(* PLC project Device (Gm2xx), 未知 HydTechnology 0.1.0.0 *)
(* stored: creationDateTime 2026-08-13T17:06:11, modificationDateTime 2026-08-15T17:48:11 *)

(* __LUBAN_DATATYPE_TEXT_META__:{"comment":"","enum_value_comments":{"FTNone":"不滤波","FTLowPass":"低通滤波","FTMedian":"中值滤波","FTLimit":"限幅滤波","FTMovingAverage":"滑动窗口均值滤波"}} *)
TYPE E_FilterType : (FTNone, FTLowPass, FTMedian, FTLimit, FTMovingAverage, FTLowPassAndMovingAverage);
END_TYPE

TYPE ST_FilterConfig : STRUCT
  eType : E_FilterType;
  rParam1 : REAL := 0.1;  (* 通用参数1: *)
  uiParam2 : UINT := 3;  (* 通用参数2: - MovingAverage: 窗口大小(采样个数) *)
END_STRUCT;
END_TYPE

TYPE ST_SensorConfig : STRUCT
  rZeroVoltage : REAL;  (* 零点电压 *)
  rMaxVoltage : REAL;  (* 最大电压 *)
  rRange : REAL;  (* 量程 (例如: 10.0 MPa 或 500.0 mm) *)
END_STRUCT;
END_TYPE

TYPE E_AxisState : (eInit, eReady, eIdle, eBusy, eDone, eStopping, eStopped, eEmergencyStop, eError);
END_TYPE

TYPE E_AxisMode : (eNone, ePosition, eVelocity, ePressure);
END_TYPE

TYPE E_PumpPolicy : (eMotionDefault, eProcessPriority);
END_TYPE

TYPE E_ProcessStep : (eStepIdle, eStepSegment1, eStepSegment2, eStepPressure, eStepDwell, eStepDone, eStepError);
END_TYPE

TYPE ST_AxisStatus : STRUCT
  eState : E_AxisState;
  bEnabled : BOOL;
  bBusy : BOOL;
  bDone : BOOL;
  bError : BOOL;
  udiErrorID : UDINT;
  rActualPosition : LREAL;
  rActualVelocity : LREAL;
  rActualPressure : REAL;
END_STRUCT;
END_TYPE

TYPE ST_HydPumpStatus : STRUCT
  rPumpSpeed : REAL;
  bConflict : BOOL;
  bBusy : BOOL;
  bDone : BOOL;
  bError : BOOL;
  wErrorID : WORD;
  bCycleReentry : BOOL;
END_STRUCT;
END_TYPE

TYPE ST_HydAxisRef : STRUCT
  bFunBlockStart : BOOL;  (* FB：启动信号 *)
  bStart : BOOL;  (* 轴：启动信号 *)
  bStop : BOOL;  (* 轴：停止信号 *)
  uiDir : UINT;  (* 轴：设定方向 *)
  udiPos : UDINT;  (* 轴：设定位置 *)
  uiSpd : UINT;  (* 轴：设定速度 *)
  uiEndSpd : UINT;  (* 轴：设定结束速度 *)
  uiPres : UINT;  (* 轴：设定压力 *)
  rPosition : REAL;  (* 轴：反馈位置 *)
  rVeloctity : REAL;  (* 轴：反馈速度 *)
  rPerssure : REAL;  (* 轴：反馈压力 *)
  rFlow : REAL;  (* 轴：反馈流量 *)
  iStep : INT;  (* 轴：反馈当前步号 *)
  rActPressure : REAL;
  rActPosition : REAL;
  rActVelocity : REAL;
  rMaxSpeed : REAL;  (* 当前轴的最大速度设定 *)
  rMaxSpeedExtend : REAL;  (* 液压轴伸出侧最大速度 *)
  rMaxSpeedRetract : REAL;  (* 液压轴缩回侧最大速度 *)
  rVelToFlowGain : REAL := 0.2;  (* 速度流量增益 *)
  rCylinderExtendArea : REAL := 0;  (* 油缸伸出腔有效面积mm2 *)
  rCylinderRetractArea : REAL := 0;  (* 油缸缩回腔有效面积mm2 *)
  iTypePressurePID : SINT := 4;  (* 压力闭环类型 *)
  iAxisID : SINT := -1;  (* 轴索引 *)
  iMechanismType : SINT := 0;  (* 机械运动学类型 *)
END_STRUCT;
END_TYPE

INTERFACE ?
END_INTERFACE

INTERFACE ?
END_INTERFACE

FUNCTION_BLOCK FB_LimitFilter
  VAR_INPUT
    rInput : REAL;
    rMaxDiff : REAL;  (* RC:[最大允许变化幅值] *)
  END_VAR
  VAR_OUTPUT
    rOutput : REAL;
  END_VAR
  VAR
    bFirstRun : BOOL := TRUE;
  END_VAR

            IF bFirstRun THEN
    rOutput := rInput;
    bFirstRun := FALSE;
ELSE
    IF ABS(rInput - rOutput) > rMaxDiff THEN
        rOutput := rOutput; // 超出限幅，保持上次值不变
    ELSE
        rOutput := rInput;  // 正常范围内，更新
    END_IF;
END_IF;
          
END_FUNCTION_BLOCK

FUNCTION_BLOCK FB_LowPassFilter
  VAR_INPUT
    rInput : REAL;
    rAlpha : REAL;  (* RC:[滤波系数 (0.0~1.0)] *)
  END_VAR
  VAR_OUTPUT
    rOutput : REAL;
  END_VAR
  VAR
    bFirstRun : BOOL := TRUE;
  END_VAR

            IF bFirstRun THEN
    rOutput := rInput;
    bFirstRun := FALSE;
ELSE
    rOutput := rOutput + rAlpha * (rInput - rOutput);
END_IF;
          
END_FUNCTION_BLOCK

FUNCTION_BLOCK FB_MedianFilter
  VAR_INPUT
    rInput : REAL;
  END_VAR
  VAR_OUTPUT
    rOutput : REAL;
  END_VAR
  VAR
    aBuffer : ARRAY[1..3] OF REAL;
    iPtr : INT := 1;
    aSort : ARRAY[1..3] OF REAL;
    i : INT;
    j : INT;
    rTemp : REAL;
  END_VAR

            // 存入循环缓冲区
aBuffer[iPtr] := rInput;
iPtr := iPtr + 1;
IF iPtr > 3 THEN iPtr := 1; END_IF;

// 复制到排序数组
aSort := aBuffer;

// 冒泡排序 (3个元素，最多3次比较)
FOR i := 1 TO 2 DO
    FOR j := 1 TO (3 - i) DO
        IF aSort[j] > aSort[j+1] THEN
            rTemp := aSort[j];
            aSort[j] := aSort[j+1];
            aSort[j+1] := rTemp;
        END_IF;
    END_FOR;
END_FOR;

// 取中间值
rOutput := aSort[2];
          
END_FUNCTION_BLOCK

FUNCTION_BLOCK FB_MovingAverageFilter
  VAR_INPUT
    rInput : REAL;
    uiSize : UINT := 1;  (* RC:[窗口大小] *)
  END_VAR
  VAR_OUTPUT
    rOutput : REAL;
  END_VAR
  VAR
    aBuffer : ARRAY[1..100] OF REAL;  (* RC:[最大支持100个数据窗口] *)
    iPtr : UINT := 1;
    rSum : REAL;
    iCount : INT := 0;
    i : UINT;
  END_VAR

            IF uiSize > 100 THEN uiSize := 100; END_IF;
IF uiSize = 0 THEN uiSize := 1; END_IF;

// 更新缓冲区
aBuffer[iPtr] := rInput;
iPtr := iPtr + 1;
IF iPtr > uiSize THEN iPtr := 1; END_IF;

// 求和计算平均值
rSum := 0.0;
FOR i := 1 TO uiSize DO
    rSum := rSum + aBuffer[i];
END_FOR;

rOutput := rSum / UINT_TO_REAL(uiSize);
          
END_FUNCTION_BLOCK

FUNCTION_BLOCK FB_PositionSensor
  VAR_INPUT
    uiRawADC : UINT;
  END_VAR
  VAR_OUTPUT
    rActualValue : REAL;  (* RC:[滤波后的最终输出] *)
    rActualValueDeriv : REAL;
    rRawValue : REAL;  (* RC:[未滤波的原始转换值 (便于调试对比)] *)
    bAlarm : BOOL;
  END_VAR
  VAR
    stConfig : ST_SensorConfig;
    stFilterCfg : ST_FilterConfig;
    rVoltage : REAL;
    fbLowPass : FB_LowPassFilter;  (* UC:[实例化滤波器] *)
    fbLimit : FB_LimitFilter;
    fbMedian : FB_MedianFilter;
    fbMovingAvg : FB_MovingAverageFilter;
    bUpperLimit : BOOL;  (* UC:[可以在此扩展位置传感器特有的变量，例如：位置限位报警] *)
    bLowerLimit : BOOL;
    rLastActualValue : REAL;
  END_VAR
  VAR CONSTANT
    cADC_MAX : REAL := 65535.0;
    cVOLTAGE_MAX : REAL := 10.0;
    cTCycle : REAL := 0.001;
  END_VAR

            // --- 主逻辑 ---

// 1. 物理量转换
IF (stConfig.rMaxVoltage - stConfig.rZeroVoltage) <= 0.0 THEN
    bAlarm := TRUE;
    rRawValue := 0.0;
ELSE
    bAlarm := FALSE;
    rRawValue := (UINT_TO_REAL(uiRawADC) - stConfig.rZeroVoltage) / 
                 (stConfig.rMaxVoltage - stConfig.rZeroVoltage) * 
                 stConfig.rRange;
    rRawValue := LIMIT(0.0,rRawValue,stConfig.rRange);
END_IF;

// 2. 滤波处理链 (采用单一配置切换，若需组合可级联调用)
CASE stFilterCfg.eType OF
    FTLowPass:
        fbLowPass(rInput := rRawValue, rAlpha := stFilterCfg.rParam1);
        rActualValue := fbLowPass.rOutput;
        
    FTLimit:
        fbLimit(rInput := rRawValue, rMaxDiff := stFilterCfg.rParam1);
        rActualValue := fbLimit.rOutput;
        
    FTMedian:
        fbMedian(rInput := rRawValue);
        rActualValue := fbMedian.rOutput;
        
    FTMovingAverage:
        fbMovingAvg(rInput := rRawValue, uiSize := stFilterCfg.uiParam2);
        rActualValue := fbMovingAvg.rOutput;
    
    FTLowPassAndMovingAverage:
        fbLowPass(rInput := rRawValue, rAlpha := stFilterCfg.rParam1);
        fbMovingAvg(rInput :=  fbLowPass.rOutput, uiSize := stFilterCfg.uiParam2);
        rActualValue := fbMovingAvg.rOutput;     
      
ELSE
    // None: 不滤波
    rActualValue := rRawValue;
END_CASE;

rActualValueDeriv := ( rActualValue - rLastActualValue )/cTCycle;
rLastActualValue := rActualValue;
          

METHOD Init : BOOL
  VAR_INPUT
    rZero : REAL;
    rMax : REAL;
    rRng : REAL;
  END_VAR
                  stConfig.rZeroVoltage := rZero;
stConfig.rMaxVoltage  := rMax;
stConfig.rRange       := rRng;
Init := TRUE;
                
END_METHOD

METHOD SetFilter : BOOL
  VAR_INPUT
    eType : E_FilterType;
    rParam1 : REAL;
    uiParam2 : UINT;
  END_VAR
                  stFilterCfg.eType := eType;
stFilterCfg.rParam1 := rParam1;
stFilterCfg.uiParam2 := uiParam2;
SetFilter := TRUE;
                
END_METHOD
END_FUNCTION_BLOCK

FUNCTION_BLOCK FB_PressureSensor
  VAR_INPUT
    uiRawADC : UINT;
  END_VAR
  VAR_OUTPUT
    rActualValue : REAL;  (* RC:[滤波后的最终输出] *)
    rRawValue : REAL;  (* RC:[未滤波的原始转换值 (便于调试对比)] *)
    bAlarm : BOOL;
  END_VAR
  VAR
    stConfig : ST_SensorConfig;
    stFilterCfg : ST_FilterConfig;
    fbLowPass : FB_LowPassFilter;  (* UC:[实例化滤波器] *)
    fbLimit : FB_LimitFilter;
    fbMedian : FB_MedianFilter;
    fbMovingAvg : FB_MovingAverageFilter;
  END_VAR
  VAR CONSTANT
    cADC_MAX : REAL := 65535.0;
    cVOLTAGE_MAX : REAL := 10.0;
  END_VAR

            
// 1. 物理量转换
IF (stConfig.rMaxVoltage - stConfig.rZeroVoltage) <= 0.0 THEN
    bAlarm := TRUE;
    rRawValue := 0.0;
ELSE
    bAlarm := FALSE;
    rRawValue := (UINT_TO_REAL(uiRawADC) - stConfig.rZeroVoltage) / 
                 (stConfig.rMaxVoltage - stConfig.rZeroVoltage) * 
                 stConfig.rRange;
    rRawValue := LIMIT(0.0,rRawValue,stConfig.rRange);

END_IF;

// 2. 滤波处理链 (采用单一配置切换，若需组合可级联调用)
CASE stFilterCfg.eType OF
    FTLowPass:
        fbLowPass(rInput := rRawValue, rAlpha := stFilterCfg.rParam1);
        rActualValue := fbLowPass.rOutput;
        
    FTLimit:
        fbLimit(rInput := rRawValue, rMaxDiff := stFilterCfg.rParam1);
        rActualValue := fbLimit.rOutput;
        
    FTMedian:
        fbMedian(rInput := rRawValue);
        rActualValue := fbMedian.rOutput;
        
    FTMovingAverage:
        fbMovingAvg(rInput := rRawValue, uiSize := stFilterCfg.uiParam2);
        rActualValue := fbMovingAvg.rOutput;

    FTLowPassAndMovingAverage:
        fbLowPass(rInput := rRawValue, rAlpha := stFilterCfg.rParam1);
        fbMovingAvg(rInput :=  fbLowPass.rOutput, uiSize := stFilterCfg.uiParam2);
        rActualValue := fbMovingAvg.rOutput;  
        
ELSE
    // None: 不滤波
    rActualValue := rRawValue;
END_CASE;
          

METHOD Init : BOOL
  VAR_INPUT
    rZero : REAL;
    rMax : REAL;
    rRng : REAL;
  END_VAR
                  stConfig.rZeroVoltage := rZero;
stConfig.rMaxVoltage  := rMax;
stConfig.rRange       := rRng;
Init := TRUE;
                
END_METHOD

METHOD SetFilter : BOOL
  VAR_INPUT
    eType : E_FilterType;
    rParam1 : REAL;
    uiParam2 : UINT;
  END_VAR
                  stFilterCfg.eType := eType;
stFilterCfg.rParam1 := rParam1;
stFilterCfg.uiParam2 := uiParam2;
SetFilter := TRUE;
                
END_METHOD
END_FUNCTION_BLOCK

FUNCTION_BLOCK FB_ServoControl
  VAR_INPUT
    StartMotor : BOOL;  (* RC:[TRUE: 使能并启动电机, FALSE: 减速停止并断使能] *)
    SetVelCmd : REAL;
    FlowRateLimit : UINT;
    uiMaxMotorSpeed : UINT;
    EnSimulation : BOOL;
    SelfLearn : BOOL;
    UsePlanner : BOOL;
    tcycle : REAL := 0.001;
  END_VAR
  VAR_OUTPUT
    ActSpeedRPM : UINT;
    ActPressBAR : UINT;
    outErrorID : UINT;
    Status : UINT;
    ActMotorPos : UINT;  (* RC:[360deg] *)
    ActTorquePercent : UINT;  (* RC:[0.1%] *)
  END_VAR
  VAR
    STATE_INIT : DINT := 0;  (* UC:[--- 状态机常量 ---] *)
    STATE_READ_SDO1 : DINT := 1;
    STATE_READ_SDO2 : DINT := 2;
    STATE_WRITE_PARAM : DINT := 10;
    STATE_SELFLEARN : DINT := 20;
    STATE_SET_MODE : DINT := 30;
    STATE_IDLE : DINT := 40;  (* RC:[等待使能] *)
    STATE_RUNNING : DINT := 50;  (* RC:[速度运行中] *)
    STATE_STOPPING : DINT := 60;  (* RC:[减速停机中] *)
    STATE_ERROR : DINT := 99;
    iState : DINT := 0;  (* UC:[--- 内部变量 ---] *)
    fbDelay : TON;  (* UC:[--- 功能块实例 ---] *)
    fbPower : MC_Power;
    fbFollowVel : SMC_FollowVelocity;
    fbSetPar : MC_WriteParameter;
    fbSetBoolPar : MC_WriteBoolParameter;
    fbReset : MC_Reset;
    fbModeCtrl : MC_SetControllerMode;
    fbReadVel : MC_ReadActualVelocity;
    fbReadPos : MC_ReadActualPosition;
    fbReadTor : MC_ReadActualTorque;
    fbSDORead : PorgaSDOUpload;
    fbStartMotorSelfLearn : StartMotorSelfLearn;
    nAxisRef : AXIS_REF := 0;
    bPowerCmd : BOOL := FALSE;  (* RC:[映射到 MC_Power.Enable] UC:[--- 运动控制核心指令标志位 ---] *)
    bMoveCmd : BOOL := FALSE;  (* RC:[映射到 SMC_FollowVelocity.Execute] *)
    dfSetVel : LREAL := 0.0;  (* RC:[映射到 SMC_FollowVelocity.Velocity] *)
    Error : BOOL := 0;  (* UC:[--- 数据与参数 ---] *)
    ErrorID : WORD := 0;
    MaxVel : LREAL := 12000.0;
    MaxAcc : LREAL := 12000.0;
    MaxJerk : LREAL := 12000.0;
    dfActVel : LREAL := 0.01;
    dfActVelFb : LREAL := 0.01;
    dfActPosFb : LREAL := 0.01;
    dfActTor : LREAL := 0.01;
    dir : LREAL := -1.0;
    fMotorSpeedLimit : LREAL := 0.0;
    fSetVel : LREAL := 0.0;
    dfMinVel : LREAL := -100.0;
    wNumBitEnc : UDINT := 0;
    wTempVar : UDINT := 0;
    dfResolutionEnc : LREAL := 0.0;
    wDirRotate : WORD := 0;
    arMotorParam : PAR_WORD_ARRAY := [3333, 107, 380, 20, 200, 5000, 100, 0, 0, 0];
  END_VAR

            
(*=====================================================================*)
(*               1. 运算与条件准备 (每周期执行)                          *)
(*=====================================================================*)

// 速度与压力设定值计算 (仅在初始化完成后计算)
IF iState >= STATE_IDLE THEN

    MaxVel  := UINT_TO_LREAL(uiMaxMotorSpeed) * (360.0/60.0); 
    MaxAcc  := 2.0 * MaxVel;
    MaxJerk := 3.0 * MaxVel;
    fMotorSpeedLimit := UINT_TO_LREAL(uiMaxMotorSpeed) * LIMIT(0, FlowRateLimit, 1000) * 0.001;
    fSetVel := REAL_TO_LREAL(SetVelCmd);
    fSetVel := LIMIT( dfMinVel, fSetVel, fMotorSpeedLimit );     
    
    fSetVel := fSetVel * dir;
END_IF;

// 使能命令统一映射 (PowerEnable 掌控全局)
bPowerCmd := StartMotor AND (iState >= STATE_IDLE);

(*=====================================================================*)
(*               2. 状态机 (仅控制逻辑流转与指令赋值)                     *)
(*=====================================================================*)

CASE iState OF

    0: // 0: 初始化IP与SDO1
        
        fbSDORead( Axis := nAxisRef, Execute := TRUE, Index := 19, Size := 1 );
        iState := STATE_READ_SDO1;

    1: // 1: 等待SDO1读取完成 (异步处理)
        fbSDORead( Axis := nAxisRef, Execute := TRUE, Index := 19, Size := 1 );
        IF fbSDORead.Done THEN
            wNumBitEnc := WORD_TO_UDINT( fbSDORead.ValueArray[1] );
            IF wNumBitEnc > 1 AND wNumBitEnc < 60 THEN
                wTempVar := SHL(1, wNumBitEnc);
            ELSE
                wTempVar := SHL(1, 12);
            END_IF;
            dfResolutionEnc := UDINT_TO_LREAL(wTempVar);
            fbSDORead( Execute := FALSE );
            fbSDORead( Axis := nAxisRef, Execute := TRUE, Index := 106, Size := 1 );
            iState := STATE_READ_SDO2;
        END_IF;

    2: // 2: 等待SDO2读取完成
        fbSDORead( Axis := nAxisRef, Execute := TRUE, Index := 106, Size := 1 );
        IF fbSDORead.Done THEN
            wDirRotate := fbSDORead.ValueArray[1];
            fbSDORead( Execute := FALSE );
            iState := STATE_WRITE_PARAM;
        END_IF;

    10: // 10: 写入参数与仿真设置
        fbSetPar(Axis := nAxisRef, Execute := TRUE, ParameterNumber:= 1003, Value := dfResolutionEnc);  // 4096
        fbSetBoolPar(Axis := nAxisRef, Execute := TRUE, ParameterNumber:= 1000, Value := EnSimulation);
        IF fbSetPar.Done AND fbSetBoolPar.Done THEN
            fbSetPar(Execute := FALSE);
            fbSetBoolPar(Execute := FALSE);
            fbReset( Axis := nAxisRef, Execute := FALSE );
            fbStartMotorSelfLearn( Axis := nAxisRef, Execute := FALSE );
            iState := STATE_SELFLEARN;
        END_IF;

    20: // 20: 自学习
        IF SelfLearn THEN
            fbStartMotorSelfLearn( Axis := nAxisRef, Execute := TRUE,
                                   ResetServoParam := TRUE, WriteServoParam := TRUE,
                                   MotorLearn := TRUE, ParameterArray := arMotorParam );
            IF fbStartMotorSelfLearn.Done THEN
                fbStartMotorSelfLearn(Execute := FALSE);
                iState := STATE_SET_MODE;
            END_IF;
        ELSE
            iState := STATE_SET_MODE;
        END_IF;

    30: // 30: 设置控制模式
        fbModeCtrl(Axis := nAxisRef, Execute := TRUE, ControllerMode := mcFollowVelocity, ExecutionMode := mcImmediately);
        IF fbModeCtrl.Done THEN
            fbModeCtrl(Execute := FALSE);
            iState := STATE_IDLE;
        END_IF;

    40: // 40: 待机状态 (等待 PowerEnable)
        bMoveCmd := FALSE;
        dfSetVel := 0.0;
        // 核心逻辑：给使能 且 电机已成功使能，则立即启动速度控制
        IF StartMotor AND fbPower.Status THEN
            iState := STATE_RUNNING;
        END_IF;

    50: // 50: 速度运行中
        bMoveCmd := TRUE;
        dfSetVel := fSetVel * (360.0/60.0); // RPM 转换 UU/s

        // 核心逻辑：一旦失去使能信号，立即进入减速停机
        IF NOT StartMotor THEN
            iState := STATE_STOPPING;
        END_IF;

    60: // 60: 减速停机中
        bMoveCmd := TRUE;  // 保持速度块 Execute，以控制减速曲线
        dfSetVel := 0.0;   // 目标速度设为 0

        // 减速中途，如果使能信号恢复，立即恢复运行
        IF StartMotor THEN
            fbDelay(IN := FALSE); // 清除停机定时器
            iState := STATE_RUNNING;
        ELSE
            // 速度低于阈值开始计时，若速度反弹则自动复位定时器
            fbDelay(IN := ABS(dfActVel) < 5.0, PT := TIME#1S);
            IF fbDelay.Q THEN
                bMoveCmd := FALSE;    // 停机完成，撤销速度控制命令
                fbDelay(IN := FALSE); // 复位定时器
                iState := STATE_IDLE; // 回到待机 (bPowerCmd随之变FALSE，自动断使能)
            END_IF;
        END_IF;

    99: // 99: 错误状态
        Error := TRUE;
        bMoveCmd := FALSE;

END_CASE;

(*=====================================================================*)
(*          3. 统一调用 PLCopen 功能块 (严格遵循规范，每周期执行)         *)
(*=====================================================================*)
//(*  更新液压系统模型 *)
//hydraulic_sys.motorvelocity := SetVelCmd;
//hydraulic_sys.tcycle := tcycle;
//hydraulic_sys.knum := 5.4;   // 4.2, 1.162, 5.4
//hydraulic_sys.ttau := 1.0;   // 0.4, 0.171, 1.0 
//hydraulic_sys.delaytime := 0.0;  // 1.0 max , 0.438
//hydraulic_sys();

// 使能控制
fbPower( Axis := nAxisRef, Enable := bPowerCmd, EnablePositive := TRUE, EnableNegative := TRUE);

// 速度跟随控制
fbFollowVel( Axis := nAxisRef, Execute := bMoveCmd, Velocity := dfSetVel);

// 反馈读取 (进入Idle后即开始读取，保证状态监控连续性)
IF iState >= STATE_IDLE THEN
    fbReadVel( Axis := nAxisRef, Enable := TRUE, Velocity => dfActVel, VelocityFeedback => dfActVelFb);
    fbReadPos( Axis := nAxisRef, Enable := TRUE, Position => dfActPosFb );
    fbReadTor( Axis := nAxisRef, Enable := TRUE, Torque   => dfActTor);  
END_IF;

// 错误捕获 (从运动功能块中提取错误)
IF fbFollowVel.Error THEN
    ErrorID := fbFollowVel.ErrorID;
    iState := STATE_ERROR;
END_IF;

(*=====================================================================*)
(*                      4. 输出映射                                     *)
(*=====================================================================*)

Status          := DINT_TO_UINT(iState);
outErrorID      := ErrorID;
ActSpeedRPM := DINT_TO_UINT( LREAL_TO_DINT(dfActVel*60.0/360.0) );
ActTorquePercent := DINT_TO_UINT( LREAL_TO_DINT(dfActTor) );
          
END_FUNCTION_BLOCK

FUNCTION_BLOCK FB_HydAxis
  VAR_IN_OUT
    stHydAxisRef : ST_HydAxisRef;
  END_VAR
  VAR_INPUT
    bStart : BOOL;
    bStop : BOOL;
    bEStop : BOOL;
    bReset : BOOL;
    uiDir : UINT;  (* RC:[0:无效 1:正向 2:反向] *)
    uiMode : UINT;  (* RC:[0:无效 1:位置 2:速度 3:压力] *)
    uiPres : UINT;
    uiSpd : UINT;
    uiEndSpd : UINT;
    udiPos : UDINT;
    uiForce : UINT;
    uiAcc : UINT;
    uiDec : UINT;
    uiJerk : UINT;
    kkk : UINT;
  END_VAR
  VAR_OUTPUT
    bBusy : BOOL;  (* RC:[TRUE=轴层当前仍保持有效执行命令] *)
    bDone : BOOL; // TRUE=位置模式下到达InEndVelocity(段结束); TRUE=非位置模式下指令执行完成且空闲;
    bInVelocity : BOOL;
    bInPressure : BOOL;
    bAlarm : BOOL;
    dwAlarmID : DWORD;
  END_VAR
  VAR
    iStep : INT;  (* RC:[0初始化, 10空闲, 100运行, 105运行过渡(产生脉冲), 200停止, 300急停, 400复位, 900报警] *)
    fbCreate : HYD_CreateMotion;
    fbMoveContAbs : HYD_MoveContinuousAbsolute;
    fbMoveVel : HYD_MoveVelocity;
    fbPresHdl : HYD_PressureHandle;
    fbStop : HYD_Stop;
    fbEStop : HYD_Stop;
    fbReset : HYD_Reset;
    fbReadFB : HYD_ReadSimFeedback;
    fbHYD_WriteParameter : HYD_WriteParameter;
    fbHYD_SetAxisFeedback : HYD_SetAxisFeedback;
    fbCalcMaxSpeed : FB_CalcAxisMaxSpeed;
    siAxisId : SINT;
    rTrigStart : R_TRIG;
    rTrigStop : R_TRIG;
    rTrigEStop : R_TRIG;
    rTrigReset : R_TRIG;
    rTrigDone : R_TRIG;
    uiActiveMode : UINT;  (* RC:[当前执行模式 (1:Pos, 2:Vel, 3:Pres)] *)
    bCmdExecute : BOOL;  (* RC:[统一控制当前活跃模式的 Execute 引脚] *)
    iDir : SINT;
    rPos : REAL;
    rVel : REAL;
    rEndVel : REAL;  (* RC:[终点速度] *)
    rPres : REAL;
    rAcc : REAL;
    rDec : REAL;
    rJerk : REAL;
    bFBError : BOOL;
    wFBErrorID : WORD;
    iDoneCnt : INT := 0;
    rMaxSpeed : REAL;  (* RC:[单位mm/s] *)
    rPosition : REAL;
    rVeloctity : REAL;
    rFlow : REAL;
    rPerssure : REAL;
    rCycle : REAL;
  END_VAR

            // 仅作监视调试使用
// 轴：启动信号、停止信号、设定位置、设定速度、设定结束速度、设定压力
stHydAxisRef.bStart := bStart;
stHydAxisRef.bStop := bStop;
stHydAxisRef.uiDir := uiDir;
stHydAxisRef.udiPos := udiPos;
stHydAxisRef.uiSpd := uiSpd;
stHydAxisRef.uiEndSpd := uiEndSpd;
stHydAxisRef.uiPres := uiPres;

//--- 1. 边沿检测 & 参数映射 ---
rTrigStart(CLK := bStart);
rTrigStop(CLK := bStop);
rTrigEStop(CLK := bEStop);
rTrigReset(CLK := bReset);
// 将Done检测移出CASE，确保全周期扫描，不错过InEndVelocity的上升沿
rTrigDone(CLK := fbMoveContAbs.InEndVelocity); 

rMaxSpeed := stHydAxisRef.rMaxSpeed;

//IF stHydAxisRef.rCylinderExtendArea > 0.0 AND stHydAxisRef.rCylinderRetractArea > 0.0 THEN
//  IF uiDir = 1 THEN
//    rMaxSpeed := stHydAxisRef.rMaxSpeedExtend;
//  ELSE
//    rMaxSpeed := stHydAxisRef.rMaxSpeedRetract;
//  END_IF;
//END_IF;

rPres := MAX(UINT_TO_REAL(uiPres), 0.0)*0.1;   //压力设定
rVel  := UINT_TO_REAL(uiSpd)*0.1*0.01*rMaxSpeed;  //速度设定
rEndVel := UINT_TO_REAL(uiEndSpd)*0.1*0.01*rMaxSpeed;  //终点速度，连续轨迹关键：设定终点速度等于最大速度，实现"到位不停车"或平滑过渡
rPos  := UDINT_TO_REAL(udiPos)*0.01;  //位置设定


IF uiAcc = 0 THEN rAcc := 200; ELSE rAcc  := rMaxSpeed/UINT_TO_REAL(uiAcc)*1000; END_IF;  
IF uiDec = 0 THEN rDec := 200; ELSE rDec  := rMaxSpeed/UINT_TO_REAL(uiDec)*1000; END_IF;  
IF uiJerk = 0 THEN rJerk := 0; ELSE rJerk := rMaxSpeed/UINT_TO_REAL(uiJerk); END_IF;

iDir := uiDir;  
//--- 2. 状态机主逻辑 ---
CASE iStep OF

    0: // 初始化
        fbCreate(USE_SIMULATION := 0, MECHANISM_TYPE:= stHydAxisRef.iMechanismType);
        IF fbCreate.DONE THEN
            siAxisId := fbCreate.AXISID;
            stHydAxisRef.iAxisID := siAxisId;
            SetVelocityToFlowGain(stHydAxisRef.rVelToFlowGain);
            SetPidType( SINT_TO_REAL(stHydAxisRef.iTypePressurePID) );
            SetCylinderConfig(stHydAxisRef.rCylinderExtendArea, stHydAxisRef.rCylinderRetractArea );
            fbCalcMaxSpeed(stHydAxisRef.rCylinderExtendArea, stHydAxisRef.rCylinderRetractArea, 1800, 50, stHydAxisRef.iMechanismType );
            stHydAxisRef.rMaxSpeedExtend  := fbCalcMaxSpeed.rMaxSpeedExtend;
            stHydAxisRef.rMaxSpeedRetract := fbCalcMaxSpeed.rMaxSpeedRetract;
            iStep := 10;
        ELSIF fbCreate.ERROR THEN
            bAlarm := TRUE; dwAlarmID := 16#00000001; iStep := 900;
        END_IF;

    10: // 空闲
        bCmdExecute := FALSE; 
        bDone := FALSE; // 重置完成信号
        IF rTrigEStop.Q THEN
            iStep := 300;
        ELSIF rTrigStop.Q THEN
            iStep := 200;
        ELSIF rTrigReset.Q AND bAlarm THEN
            iStep := 400;
        ELSIF rTrigStart.Q AND uiMode >= 1 AND uiMode <= 3 THEN
            uiActiveMode := uiMode; 
            bCmdExecute := TRUE; // 启动时直接置高
            iStep := 100;           
        END_IF;

    100: // 运行中
        // 默认保持执行状态
        bCmdExecute := TRUE; 
        
        // 1. 错误监测 (所有模式通用)
        CASE uiActiveMode OF
            1: bFBError := fbMoveContAbs.ERROR; wFBErrorID := fbMoveContAbs.ERRORID;
            2: bFBError := fbMoveVel.ERROR; wFBErrorID := fbMoveVel.ERRORID;
            3: bFBError := fbPresHdl.ERROR; wFBErrorID := fbPresHdl.ERRORID;
        END_CASE;
        
        IF bFBError THEN
            bAlarm := TRUE; dwAlarmID := wFBErrorID; iStep := 900;
            
        // 2. 段切换触发 (核心逻辑)
        ELSIF rTrigStart.Q THEN
            // 检测到新的启动信号
            IF uiMode = uiActiveMode THEN
                // 同模式重触发（例如射胶第一段->第二段）：
                // 进入过渡步，拉低Execute，下一周期再拉高，产生上升沿
                iStep := 105; 
            ELSIF uiMode >= 1 AND uiMode <= 3 THEN
                // 跨模式切换（如位置->压力）：直接更改模式
                // 注意：有些运动控制库需要Stop才能切换模式，这里假设支持无缝切换或由BufferMode处理
                uiActiveMode := uiMode; 
                // 如果库不支持直接修改参数切换，此处也应跳转Step 105
            END_IF;
        END_IF;
        
        // 3. 中断监测
        IF rTrigEStop.Q THEN iStep := 300;
        ELSIF rTrigStop.Q THEN iStep := 200;
        END_IF;

    105: // 运行过渡步 (产生Execute脉冲)
        // 此步仅保持1个周期
        bCmdExecute := FALSE; // 拉低Execute
        bDone := FALSE;      // 清除上一段的完成标志
        iStep := 100;        // 立即回100，在100中bCmdExecute变TRUE，形成上升沿

    200: // 正常停止
        fbStop(AXISID := siAxisId, EXECUTE := TRUE, DECELERATION := rDec); // 这里的Execute通常需要脉冲或持续，视具体FB而定，假设持续
        IF fbStop.DONE THEN
            fbStop(EXECUTE := FALSE); // 停止命令需复位
            iStep := 10;
        ELSIF fbStop.ERROR THEN
            bAlarm := TRUE; dwAlarmID := fbStop.ERRORID; iStep := 900;
        END_IF;

    300: // 急停
        fbEStop(AXISID := siAxisId, EXECUTE := TRUE, DECELERATION := 99999.0);
        IF fbEStop.DONE OR fbEStop.ERROR THEN
            fbEStop(EXECUTE := FALSE);
            bAlarm := TRUE; dwAlarmID := 16#0000FFFF; iStep := 900;
        END_IF;

    400: // 报警复位
        fbReset(AXISID := siAxisId, EXECUTE := TRUE);
        IF fbReset.DONE THEN
            fbReset(EXECUTE := FALSE);
            bAlarm := FALSE; dwAlarmID := 0; iStep := 10;
        ELSIF fbReset.ERROR THEN
            bAlarm := TRUE; dwAlarmID := fbReset.ERRORID; iStep := 900;
        END_IF;

    900: // 报警等待
        IF rTrigReset.Q THEN
            iStep := 400;
        END_IF;

END_CASE;

//--- 3. 底层 FB 统一调用区 ---
// 注意：fbStop, fbEStop, fbReset的调用已在State中处理或者在这里根据iStep统一处理
// 为了代码清晰，建议持续调用，EXECUTE由状态控制
// 但为了符合原代码结构，下面保留原风格，修正MoveContinuousAbsolute的参数

// Create 只在Init或Reset时调用一次即可，原代码持续调用没问题(内部有Enable管理)
// fbCreate(...); 
rCycle := rCycle + 0.001;
fbHYD_SetAxisFeedback(
     AXISID := siAxisId,
     ENABLE := 1,
     ACT_POSITION := stHydAxisRef.rActPosition,
     ACT_VELOCITY := stHydAxisRef.rVeloctity,
     ACT_FLOW := 0,
     ACT_PRESSURE := stHydAxisRef.rActPressure,
     TIMESTAMP := rCycle
   );

fbMoveContAbs(
    AXISID := siAxisId, 
    EXECUTE := (uiActiveMode = 1) AND bCmdExecute, 
    POSITION := rPos, 
    VELOCITY := rVel,
    ENDVELOCITY := rEndVel,    // 关键修改：设定终点速度，保证InEndVelocity能正常触发
    ENDVELOCITYDIRECTION := iDir, // 0=Current/Positive, 需根据实际情况设定
    ACCELERATION := rAcc, 
    DECELERATION := rDec, 
    JERK := rJerk, 
    DIRECTION := iDir,
    ADAPTENDVELTOAVOIDOVERSHOOT := TRUE,
    PRESSURELIMIT := rPres
    // BufferMode 可根据库支持情况添加，若不支持则依靠Step 105的脉冲机制
);



fbMoveVel(
    AXISID := siAxisId, EXECUTE := (uiActiveMode = 2) AND bCmdExecute, 
    CONTINUOUSUPDATE := TRUE, VELOCITY := rVel,
    ACCELERATION := rAcc, DECELERATION := rDec, JERK := rJerk, DIRECTION := iDir, BUFFERMODE := 0,PRESSURELIMIT := rPres);

fbPresHdl(
    AXISID := siAxisId, EXECUTE := (uiActiveMode = 3) AND bCmdExecute, 
    CONTINUOUSUPDATE := TRUE, PRESSURE := rPres, PRESSURERAMPRATE := rAcc, DURATION := 0.0, BUFFERMODE := 0);

// Stop/EStop/Reset 需要特殊处理Execute信号，防止一直给TRUE
// 修改为根据状态决定EXECUTE
IF iStep = 200 THEN
    fbStop(AXISID := siAxisId, EXECUTE := TRUE, DECELERATION := rDec);
ELSE
    fbStop(AXISID := siAxisId, EXECUTE := FALSE, DECELERATION := rDec);
END_IF;

IF iStep = 300 THEN
    fbEStop(AXISID := siAxisId, EXECUTE := TRUE, DECELERATION := 99999.0);
ELSE
    fbEStop(AXISID := siAxisId, EXECUTE := FALSE, DECELERATION := 99999.0);
END_IF;

IF iStep = 400 THEN
    fbReset(AXISID := siAxisId, EXECUTE := TRUE);
ELSE
    fbReset(AXISID := siAxisId, EXECUTE := FALSE);
END_IF;

// 仅作监视调试使用
// 轴：反馈位置、反馈速度、反馈流量、反馈压力、反馈当前步号
fbReadFB(AXISID := siAxisId, ENABLE := TRUE);
IF fbReadFB.VALID THEN
    stHydAxisRef.rPosition  := fbReadFB.POSITION;
    stHydAxisRef.rVeloctity := fbReadFB.VELOCITY;
    stHydAxisRef.rFlow      := fbReadFB.FLOW;
    stHydAxisRef.rPerssure  := fbReadFB.PRESSURE;
END_IF;
//引出iStep状态
stHydAxisRef.iStep := iStep;
//--- 4. 状态输出汇总 ---
IF iStep = 10 THEN
    bBusy := FALSE; 
    bDone := FALSE; // 空闲状态下没有完成信号
ELSIF iStep = 100 OR iStep = 105 THEN
    bBusy := TRUE;  // 忙
    
    // 区分模式的Done信号
    IF uiActiveMode = 1 THEN
        // 位置模式：InEndVelocity TRUE 表示当前段已到达且速度吻合，可以进行下一段
        bDone := fbMoveContAbs.InEndVelocity; 
    ELSIF uiActiveMode = 2 THEN
        // 速度模式：通常持续运行，除非有特定停止条件，这里暂不输出Done，或根据是否达到速度判定
        bDone := fbMoveVel.InVelocity; 
    ELSIF uiActiveMode = 3 THEN
        // 压力模式
        bDone := fbPresHdl.INPRESSURE;
    ELSE
        bDone := FALSE;
    END_IF;
    
    bInVelocity := fbMoveVel.InVelocity;
    bInPressure := fbPresHdl.INPRESSURE;
    
ELSIF iStep = 200 THEN
    bBusy := TRUE; bDone := FALSE;
ELSIF iStep = 300 THEN
    bBusy := TRUE; bDone := FALSE;
ELSIF iStep = 400 THEN  
    bBusy := TRUE; bDone := FALSE;
ELSE // 900 等
    bBusy := FALSE; bDone := FALSE;
END_IF;

//TraceVariable( INDEX := 0,   VALUE := rPosition );
//TraceVariable( INDEX := 1,   VALUE := rVeloctity );




          

METHOD SetVelocityToFlowGain : BOOL
  VAR_INPUT
    rVelToFlowGain : REAL;
  END_VAR
  VAR CONSTANT
    iParamterIndex : INT := 5;
  END_VAR
                  fbHYD_WriteParameter( AXISID := siAxisId, EXECUTE := FALSE);
fbHYD_WriteParameter( AXISID := siAxisId, EXECUTE := TRUE,
                      PARAMETERNUMBER := iParamterIndex, VALUE := REAL_TO_LREAL(rVelToFlowGain) );

SetVelocityToFlowGain := fbHYD_WriteParameter.Done;
                
END_METHOD

METHOD SetPidType : BOOL
  VAR_INPUT
    rTypePID : REAL;
  END_VAR
  VAR CONSTANT
    iParamterIndex : INT := 25;
  END_VAR
                  fbHYD_WriteParameter( AXISID := siAxisId, EXECUTE := FALSE);
fbHYD_WriteParameter( AXISID := siAxisId, EXECUTE := TRUE,
                      PARAMETERNUMBER := iParamterIndex, VALUE := REAL_TO_LREAL(rTypePID) );
SetPidType := fbHYD_WriteParameter.Done;

                
END_METHOD

METHOD SetCylinderConfig : BOOL
  VAR_INPUT
    rExtendArea : REAL;
    rRetractArea : REAL;
  END_VAR
  VAR CONSTANT
    iCylinderExtendArea : INT := 31;
    iCylinderRetractArea : INT := 32;
  END_VAR
                  fbHYD_WriteParameter( AXISID := siAxisId, EXECUTE := FALSE);
fbHYD_WriteParameter( AXISID := siAxisId, EXECUTE := TRUE,
                      PARAMETERNUMBER := iCylinderExtendArea, VALUE := REAL_TO_LREAL(rExtendArea) );

SetCylinderConfig := fbHYD_WriteParameter.Done;

IF NOT SetCylinderConfig THEN
  RETURN;
END_IF;

fbHYD_WriteParameter( AXISID := siAxisId, EXECUTE := FALSE);
fbHYD_WriteParameter( AXISID := siAxisId, EXECUTE := TRUE,
                      PARAMETERNUMBER := iCylinderRetractArea, VALUE := REAL_TO_LREAL(rRetractArea) );


SetCylinderConfig := fbHYD_WriteParameter.Done;
                
END_METHOD
END_FUNCTION_BLOCK

PROGRAM program0
  VAR
    stHydAxisRef : ST_HydAxisRef;
    stElectricAxisRef : AXIS_REF;
    fbHydraulicAxis : FB_HydraulicAxis;
    fbElectricAxis : FB_ElectricAxis;
    fbTechnology : FB_HydTechnology;
    iHydraulicAxis : IHydraulicAxis;
    iElectricAxis : IAxis;
    bInitialized : BOOL;
    bMachineEnable : BOOL;
    bHydraulicRun : BOOL;
    bElectricRun : BOOL;
    bClampCommand : BOOL;
    bInjectionCommand : BOOL;
    rHydraulicVelocity : LREAL;
    rElectricVelocity : LREAL;
  END_VAR

            
(* Application smoke example. No pump request or servo arbitration is visible here. *)
IF NOT bInitialized THEN
    stHydAxisRef.iAxisID := -1;
    bMachineEnable := TRUE;
    bHydraulicRun := FALSE;
    bElectricRun := FALSE;
    rHydraulicVelocity := 20.0;
    rElectricVelocity := 1200.0;
    bInitialized := TRUE;
END_IF;

(* Both adapters expose the same common command names. *)
fbHydraulicAxis(
    stHydAxisRef := stHydAxisRef,
    bEnable := bMachineEnable,
    bMove := bHydraulicRun,
    rVelocity := rHydraulicVelocity,
    bStop := FALSE,
    bEStop := FALSE,
    bReset := FALSE,
    uiDir := 1,
    uiMode := 2,
    uiSpd := LREAL_TO_UINT(ABS(rHydraulicVelocity)),
    udiPos := 0);

fbElectricAxis(
    AxisRef := stElectricAxisRef,
    bEnable := bMachineEnable,
    bMove := bElectricRun,
    rVelocity := rElectricVelocity);

(* OOP registration boundary; concrete-to-interface assignment is handled by the target compiler. *)
iHydraulicAxis := fbHydraulicAxis;
iElectricAxis := fbElectricAxis;
fbTechnology(
    iHydraulicAxis := iHydraulicAxis,
    iElectricAxis := iElectricAxis,
    bEnable := bMachineEnable,
    ePumpPolicy := eMotionDefault,
    bAllowNegative := FALSE,
    uiMaxMotorSpeed := 1800,
    bRegisterHydraulicAxis := bInitialized,
    bRegisterElectricAxis := bInitialized,
    bClampExecute := bClampCommand,
    bInjectionExecute := bInjectionCommand);

          
END_PROGRAM

FUNCTION_BLOCK FB_CalcAxisMaxSpeed
  VAR_INPUT
    rAreaExtendSide : REAL;  (* UC:[油缸参数：无杆腔侧面积 (单位修改为: mm²)] *)
    rAreaRetractSide : REAL;  (* UC:[油缸参数：有杆腔侧面积 (单位修改为: mm²)] *)
    rPumpMaxRPM : REAL := 1800;  (* UC:[油泵参数：最大转速 (单位: rpm)] *)
    rPumpDisplacement : REAL := 50;  (* UC:[油泵参数：排量 (单位: cc/rev)] *)
    iMechanismType : SINT := 0;
  END_VAR
  VAR_OUTPUT
    rMaxSpeedExtend : REAL;  (* UC:[计算结果：伸出方向最大速度 (单位: mm/s)] *)
    rMaxSpeedRetract : REAL;  (* UC:[计算结果：缩回方向最大速度 (单位: mm/s)] *)
    bValid : BOOL;  (* UC:[状态位：计算是否有效 (用于错误指示)] *)
  END_VAR
  VAR
    rMaxFlowRate_cc : REAL;  (* UC:[中间变量：油泵最大流量 (单位: cc/min)] *)
    rCoeff : REAL := 16.667;  (* UC:[系数：从流量转换到速度的系数] *)
    rKVelocityRateExtend : REAL := 0.73;  (* RC:[曲肘开模变速比] *)
    rKVelocityRateRetract : REAL := 1.18;  (* RC:[曲肘合模变速比] *)
  END_VAR

            
// 1. 默认状态为无效
bValid := FALSE;

// 2. 参数有效性检查 (面积必须大于0，防止除零)
IF (rAreaExtendSide <= 0.0) OR (rAreaRetractSide <= 0.0) OR 
   (rPumpMaxRPM < 0.0) OR (rPumpDisplacement <= 0.0) THEN
    
    rMaxSpeedExtend  := 0.0;
    rMaxSpeedRetract := 0.0;
    
ELSE
    bValid := TRUE;

    // 3. 计算油泵最大流量
    // 结果单位为 cc/min (立方厘米/分)=mL/min
    rMaxFlowRate_cc := rPumpDisplacement * rPumpMaxRPM;

    // 4. 计算伸出最大速度
    // 公式: (流量 cc/min * 1000) / (面积 mm² * 60)
    // 简化为: 流量 * 16.667 / 面积
    rMaxSpeedExtend := (rMaxFlowRate_cc * rCoeff) / rAreaExtendSide;

    // 5. 计算缩回最大速度
    rMaxSpeedRetract := (rMaxFlowRate_cc * rCoeff) / rAreaRetractSide;

    IF iMechanismType = 1 THEN
      rMaxSpeedExtend  := rMaxSpeedExtend * rKVelocityRateExtend; // kv=f(Xm),变速比是动模板位置的函数
      rMaxSpeedRetract := rMaxSpeedRetract * rKVelocityRateRetract;
    END_IF;
END_IF;

          
END_FUNCTION_BLOCK

FUNCTION_BLOCK FB_EleAxis
  VAR
    NewLocalVar0 : DINT;
  END_VAR

            NewLocalVar0 := NewLocalVar0 + 1; 


          
END_FUNCTION_BLOCK

FUNCTION_BLOCK IAxis
  VAR_OUTPUT
    bEnabled : BOOL;
    bBusy : BOOL;
    bDone : BOOL;
    bError : BOOL;
    eState : E_AxisState;
    stStatus : ST_AxisStatus;
  END_VAR

(* IAxis contract: Enable, MoveVelocity, MoveAbsolute, Stop, EStop, Reset, Cyclic and status properties. *)
END_FUNCTION_BLOCK

FUNCTION_BLOCK IHydraulicAxis
  VAR_OUTPUT
    rRequestedFlow : REAL;
    bPumpConflict : BOOL;
  END_VAR

(* IHydraulicAxis extends IAxis and adds pressure/flow status methods. *)
END_FUNCTION_BLOCK

FUNCTION_BLOCK FB_AxisBase
  VAR_INPUT
    bEnable : BOOL;
    bEStop : BOOL;
    bReset : BOOL;
  END_VAR
  VAR_OUTPUT
    bEnabled : BOOL;
    bBusy : BOOL;
    bDone : BOOL;
    bError : BOOL;
    eState : E_AxisState;
  END_VAR
  VAR
    iState : INT;
  END_VAR

IF bEStop THEN
    iState := 7;
ELSIF bReset THEN
    iState := 0;
ELSIF bEnable THEN
    iState := 2;
ELSE
    iState := 1;
END_IF;
bEnabled := bEnable AND NOT bEStop;
bBusy := FALSE;
bDone := FALSE;
bError := (iState = 99);
END_FUNCTION_BLOCK

FUNCTION_BLOCK FB_ElectricAxis
  VAR_IN_OUT
    AxisRef : AXIS_REF;
  END_VAR
  VAR_INPUT
    bEnable : BOOL;
    bMove : BOOL;
    rVelocity : LREAL;
  END_VAR
  VAR_OUTPUT
    bEnabled : BOOL;
    bBusy : BOOL;
    bDone : BOOL;
    bError : BOOL;
    eState : E_AxisState;
    stStatus : ST_AxisStatus;
    udiErrorID : UDINT;
  END_VAR
  VAR
    fbPower : MC_Power;
    fbFollowVelocity : SMC_FollowVelocity;
  END_VAR

fbPower(Axis := AxisRef, Enable := bEnable, EnablePositive := TRUE, EnableNegative := TRUE);
fbFollowVelocity(Axis := AxisRef, Execute := bMove, Velocity := rVelocity);
bEnabled := fbPower.Status;
bBusy := fbFollowVelocity.Busy;
bDone := NOT fbFollowVelocity.Busy AND NOT fbFollowVelocity.Error AND bMove;
bError := fbPower.Error OR fbFollowVelocity.Error;
udiErrorID := WORD_TO_UDINT(fbFollowVelocity.ErrorID);
IF bError THEN
    eState := eError;
ELSIF bBusy THEN
    eState := eBusy;
ELSIF bEnabled THEN
    eState := eReady;
ELSE
    eState := eIdle;
END_IF;
stStatus.eState := eState;
stStatus.bEnabled := bEnabled;
stStatus.bBusy := bBusy;
stStatus.bDone := bDone;
stStatus.bError := bError;
stStatus.udiErrorID := udiErrorID;
END_FUNCTION_BLOCK

FUNCTION_BLOCK FB_HydraulicAxis
  VAR_IN_OUT
    stHydAxisRef : ST_HydAxisRef;
  END_VAR
  VAR_INPUT
    bEnable : BOOL;
    bMove : BOOL;
    rVelocity : LREAL;
    bStart : BOOL;
    bStop : BOOL;
    bEStop : BOOL;
    bReset : BOOL;
    uiMode : UINT;
    uiDir : UINT;
    uiSpd : UINT;
    udiPos : UDINT;
    uiPres : UINT;
  END_VAR
  VAR_OUTPUT
    bEnabled : BOOL;
    bBusy : BOOL;
    bDone : BOOL;
    bError : BOOL;
    eState : E_AxisState;
    stStatus : ST_AxisStatus;
    rRequestedFlow : REAL;
    bPumpConflict : BOOL;
    udiErrorID : UDINT;
  END_VAR
  VAR
    fbLegacyHydAxis : FB_HydAxis;
    fbReadStatus : HYD_ReadStatus;
  END_VAR

fbLegacyHydAxis(
    stHydAxisRef := stHydAxisRef,
    bStart := bStart OR bEnable OR bMove,
    bStop := bStop,
    bEStop := bEStop,
    bReset := bReset,
    uiDir := uiDir,
    uiMode := SEL(bMove OR bEnable, 2, uiMode),
    uiPres := uiPres,
    uiSpd := SEL(bMove OR bEnable, LREAL_TO_UINT(ABS(rVelocity)), uiSpd),
    udiPos := udiPos);
fbReadStatus(AXISID := stHydAxisRef.iAxisID, ENABLE := TRUE);
bBusy := fbLegacyHydAxis.bBusy;
bDone := fbLegacyHydAxis.bDone;
bError := fbLegacyHydAxis.bAlarm OR fbReadStatus.ERROR;
bEnabled := (stHydAxisRef.iAxisID >= 0) AND NOT bError;
udiErrorID := DWORD_TO_UDINT(fbLegacyHydAxis.dwAlarmID);
rRequestedFlow := fbReadStatus.REQUESTEDFLOW;
bPumpConflict := fbReadStatus.PUMPSPEEDLIMITACTIVE OR fbReadStatus.FLOWLIMITACTIVE;
IF bError THEN
    eState := eError;
ELSIF bBusy THEN
    eState := eBusy;
ELSIF bEnabled THEN
    eState := eReady;
ELSE
    eState := eIdle;
END_IF;
stStatus.eState := eState;
stStatus.bEnabled := bEnabled;
stStatus.bBusy := bBusy;
stStatus.bDone := bDone;
stStatus.bError := bError;
stStatus.udiErrorID := udiErrorID;
stStatus.rActualPressure := INT_TO_REAL(fbReadStatus.PRESSURECONTROLLERAPPLIED);
stStatus.rActualPosition := REAL_TO_LREAL(fbReadStatus.ACTUATORPOSITION);
stStatus.rActualVelocity := REAL_TO_LREAL(fbReadStatus.ACTUATORVELOCITYCOMMAND);
END_FUNCTION_BLOCK

FUNCTION_BLOCK FB_HydPumpManager
  VAR_INPUT
    bEnable : BOOL;
    ePolicy : E_PumpPolicy;
    bAllowNegative : BOOL;
    uiMaxMotorSpeed : UINT;
  END_VAR
  VAR_OUTPUT
    stStatus : ST_HydPumpStatus;
  END_VAR
  VAR
    aHydAxis : ARRAY[0..15] OF IHydraulicAxis;
    aHydAxisUsed : ARRAY[0..15] OF BOOL;
    uiHydAxisCount : UINT;
    bCycleExecuted : BOOL;
    udiCycleSequence : UDINT;
    siStrategy : SINT;
    fbGetPumpRequest : HYD_GetPumpRequest;
    fbServoControl : FB_ServoControl;
  END_VAR

IF bCycleExecuted THEN
    stStatus.bCycleReentry := TRUE;
    RETURN;
END_IF;
stStatus.bCycleReentry := FALSE;
bCycleExecuted := TRUE;
udiCycleSequence := udiCycleSequence + 1;

CASE ePolicy OF
    eMotionDefault: siStrategy := 0;
    eProcessPriority: siStrategy := 1;
ELSE
    siStrategy := 0;
END_CASE;
fbGetPumpRequest(ENABLE := bEnable, STRATEGY := siStrategy, ALLOW_NEGATIVE := bAllowNegative);
fbServoControl(StartMotor := bEnable AND NOT fbGetPumpRequest.ERROR AND NOT fbGetPumpRequest.CONFLICT, SetVelCmd := fbGetPumpRequest.PUMPSPEED, FlowRateLimit := 1000, uiMaxMotorSpeed := uiMaxMotorSpeed, EnSimulation := FALSE, SelfLearn := FALSE, UsePlanner := FALSE);
stStatus.rPumpSpeed := fbGetPumpRequest.PUMPSPEED;
stStatus.bConflict := fbGetPumpRequest.CONFLICT;
stStatus.bBusy := fbGetPumpRequest.BUSY;
stStatus.bDone := fbGetPumpRequest.DONE;
stStatus.bError := fbGetPumpRequest.ERROR;
stStatus.wErrorID := fbGetPumpRequest.ERRORID;
bCycleExecuted := FALSE;
END_FUNCTION_BLOCK

FUNCTION_BLOCK FB_ClampProcess
  VAR_INPUT
    bExecute : BOOL;
  END_VAR
  VAR_OUTPUT
    bBusy : BOOL;
    bDone : BOOL;
    bError : BOOL;
  END_VAR
  VAR
    iStep : INT;
  END_VAR

IF bExecute THEN
    bBusy := TRUE;
    bDone := FALSE;
    CASE iStep OF
        0:   iStep := 10; (* 锁模：快速接近 *)
        10:  iStep := 20; (* 锁模：低速合模 *)
        20:  iStep := 30; (* 锁模：压力建立 *)
        30:  iStep := 100; (* 锁模完成 *)
    END_CASE;
ELSE
    bBusy := FALSE;
    bDone := (iStep = 100);
END_IF;
END_FUNCTION_BLOCK

FUNCTION_BLOCK FB_MoldOpenProcess
  VAR_INPUT
    bExecute : BOOL;
  END_VAR
  VAR_OUTPUT
    bBusy : BOOL;
    bDone : BOOL;
    bError : BOOL;
  END_VAR
  VAR
    iStep : INT;
  END_VAR

IF bExecute THEN
    bBusy := TRUE;
    bDone := FALSE;
    CASE iStep OF
        0:   iStep := 10; (* 开模：脱模/破闸 *)
        10:  iStep := 20; (* 开模：快速打开 *)
        20:  iStep := 100; (* 开模：末端低速定位完成 *)
    END_CASE;
ELSE
    bBusy := FALSE;
    bDone := (iStep = 100);
END_IF;
END_FUNCTION_BLOCK

FUNCTION_BLOCK FB_InjectionProcess
  VAR_INPUT
    bExecute : BOOL;
  END_VAR
  VAR_OUTPUT
    bBusy : BOOL;
    bDone : BOOL;
    bError : BOOL;
  END_VAR
  VAR
    iStep : INT;
  END_VAR

IF bExecute THEN
    bBusy := TRUE;
    bDone := FALSE;
    CASE iStep OF
        0:   iStep := 10; (* 射胶：高速段 *)
        10:  iStep := 20; (* 射胶：低速段 *)
        20:  iStep := 30; (* 射胶：速度/压力切换 *)
        30:  iStep := 100; (* 射胶：保压结束 *)
    END_CASE;
ELSE
    bBusy := FALSE;
    bDone := (iStep = 100);
END_IF;
END_FUNCTION_BLOCK

FUNCTION_BLOCK FB_ChargeProcess
  VAR_INPUT
    bExecute : BOOL;
  END_VAR
  VAR_OUTPUT
    bBusy : BOOL;
    bDone : BOOL;
    bError : BOOL;
  END_VAR
  VAR
    iStep : INT;
  END_VAR

IF bExecute THEN
    bBusy := TRUE;
    bDone := FALSE;
    CASE iStep OF
        0:   iStep := 10; (* 储料：塑化/计量 *)
        10:  iStep := 100;
    END_CASE;
ELSE
    bBusy := FALSE;
    bDone := (iStep = 100);
END_IF;
END_FUNCTION_BLOCK

FUNCTION_BLOCK FB_EjectProcess
  VAR_INPUT
    bExecute : BOOL;
  END_VAR
  VAR_OUTPUT
    bBusy : BOOL;
    bDone : BOOL;
    bError : BOOL;
  END_VAR
  VAR
    iStep : INT;
    fbHold : TON;
  END_VAR

IF bExecute THEN
    bBusy := TRUE;
    bDone := FALSE;
    CASE iStep OF
        0:   iStep := 10; (* 顶针：前进 *)
        10:  fbHold(IN := TRUE, PT := T#500ms); (* 顶针：保压/停留 *)
        20:  iStep := 100; (* 顶针：返回完成 *)
        100: bDone := TRUE;
    END_CASE;
    IF fbHold.Q THEN
        fbHold(IN := FALSE);
        iStep := 20;
    END_IF;
ELSE
    fbHold(IN := FALSE);
    bBusy := FALSE;
    bDone := (iStep = 100);
END_IF;
END_FUNCTION_BLOCK

FUNCTION_BLOCK FB_HydTechnology
  VAR_IN_OUT
    iHydraulicAxis : IHydraulicAxis;
    iElectricAxis : IAxis;
  END_VAR
  VAR_INPUT
    bEnable : BOOL;
    ePumpPolicy : E_PumpPolicy;
    bAllowNegative : BOOL;
    uiMaxMotorSpeed : UINT;
    bRegisterHydraulicAxis : BOOL;
    bRegisterElectricAxis : BOOL;
    bClampExecute : BOOL;
    bMoldOpenExecute : BOOL;
    bInjectionExecute : BOOL;
    bChargeExecute : BOOL;
    bEjectExecute : BOOL;
  END_VAR
  VAR_OUTPUT
    bInitialized : BOOL;
    bBusy : BOOL;
    bError : BOOL;
    stPumpStatus : ST_HydPumpStatus;
  END_VAR
  VAR
    aAxis : ARRAY[0..31] OF IAxis;
    aAxisUsed : ARRAY[0..31] OF BOOL;
    uiAxisCount : UINT;
    aHydAxis : ARRAY[0..15] OF IHydraulicAxis;
    aHydAxisUsed : ARRAY[0..15] OF BOOL;
    uiHydAxisCount : UINT;
    bHydraulicRegistered : BOOL;
    bElectricRegistered : BOOL;
    fbClamp : FB_ClampProcess;
    fbMoldOpen : FB_MoldOpenProcess;
    fbInjection : FB_InjectionProcess;
    fbCharge : FB_ChargeProcess;
    fbEject : FB_EjectProcess;
    fbPumpManager : FB_HydPumpManager;
  END_VAR

IF bRegisterHydraulicAxis AND NOT bHydraulicRegistered AND (uiHydAxisCount < 16) THEN
    aHydAxis[uiHydAxisCount] := iHydraulicAxis;
    aHydAxisUsed[uiHydAxisCount] := TRUE;
    bHydraulicRegistered := TRUE;
    uiHydAxisCount := uiHydAxisCount + 1;
END_IF;
IF bRegisterElectricAxis AND NOT bElectricRegistered AND (uiAxisCount < 32) THEN
    aAxis[uiAxisCount] := iElectricAxis;
    aAxisUsed[uiAxisCount] := TRUE;
    bElectricRegistered := TRUE;
    uiAxisCount := uiAxisCount + 1;
END_IF;

fbClamp(bExecute := bClampExecute);
fbMoldOpen(bExecute := bMoldOpenExecute);
fbInjection(bExecute := bInjectionExecute);
fbCharge(bExecute := bChargeExecute);
fbEject(bExecute := bEjectExecute);
fbPumpManager(bEnable := bEnable, ePolicy := ePumpPolicy, bAllowNegative := bAllowNegative, uiMaxMotorSpeed := uiMaxMotorSpeed);
bInitialized := TRUE;
bBusy := fbPumpManager.stStatus.bBusy;
bError := fbPumpManager.stStatus.bError;
stPumpStatus := fbPumpManager.stStatus;
END_FUNCTION_BLOCK

CONFIGURATION config
  RESOURCE resource1 ON PLC
    TASK task0(INTERVAL := T#20ms, PRIORITY := 0);
    PROGRAM instance0 WITH task0 : program0;
  END_RESOURCE
END_CONFIGURATION
